SYSTEM TANK_MVCL (* Level Control System Model+View+Control+HMI *)
  (* Standard: 61499-1; Classification: Simulation; ApplicationDomain: Process Control *)
  (* Version 0.4, 2007-08-17, JHC, Holobloc Inc, Added SETUP delays for models & controller, changed AUTO tag to MODE. *)
  (* Version 0.3, 2007-08-15, JHC, Holobloc Inc, Removed space in literal "t#250 ms" *)
  (* Version 0.2, 2007-01-09, JHC, Holobloc Inc, Added tag comments. *)
  (* Version 0.1, 2004-09-13, JHC, Rockwell Automation, Extended from TANK_MVL. *)
  (* Version 0.0, 2004-09-03, JHC, Rockwell Automation, Extended from TANK_MVL. *)
  APPLICATION TANK_CTL (* Tank Control Application *)
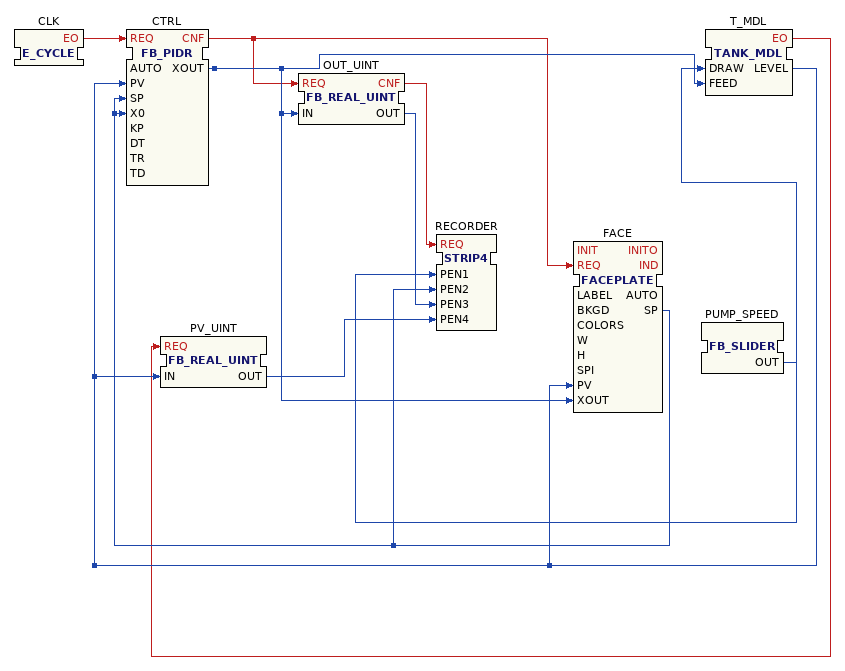
    FBS
      FACE : FACEPLATE;
      CTRL : FB_PIDR;
      RECORDER : STRIP4;
      CLK : E_CYCLE;
      T_MDL : TANK_MDL;
      PUMP_SPEED : FB_SLIDER;
      OUT_UINT : FB_REAL_UINT;
      PV_UINT : FB_REAL_UINT;
    END_FBS
    EVENT_CONNECTIONS
      CLK.EO TO CTRL.REQ;
      CTRL.CNF TO OUT_UINT.REQ;
      T_MDL.EO TO PV_UINT.REQ;
      OUT_UINT.CNF TO RECORDER.REQ;
      CTRL.CNF TO FACE.REQ;
    END_CONNECTIONS
    DATA_CONNECTIONS
      FACE.SP TO CTRL.SP;
      FACE.SP TO CTRL.X0;
      PUMP_SPEED.OUT TO T_MDL.DRAW;
      CTRL.XOUT TO T_MDL.FEED;
      T_MDL.LEVEL TO CTRL.PV;
      T_MDL.LEVEL TO FACE.PV;
      CTRL.XOUT TO FACE.XOUT;
      PUMP_SPEED.OUT TO RECORDER.PEN1;
      FACE.SP TO RECORDER.PEN2;
      CTRL.XOUT TO OUT_UINT.IN;
      OUT_UINT.OUT TO RECORDER.PEN3;
      T_MDL.LEVEL TO PV_UINT.IN;
      PV_UINT.OUT TO RECORDER.PEN4;
    END_CONNECTIONS
  END_APPLICATION
  DEVICE HMI : FRAME_DEVICE(BOUNDS := [240,100,210,270])
    RESOURCE RECORDER : PANEL_RESOURCE
      FBS
        PUMP_SPEED : SUBL_1;
        PV : SUBL_1; (* Measured (Process) Variable *)
        OUT : SUBL_1; (* Manipulated (Output) Variable *)
        RECORDER : STRIP4(COLORS := [red,orange,green,blue], BKGD := COLOR#lightGray, SIZE := [200,150], DX := 1);
        PV_UINT : FB_REAL_UINT;
        OUT_UINT : FB_REAL_UINT;
        SP : SUBL_1; (* Set Point *)
      END_FBS
      EVENT_CONNECTIONS
        PV.IND TO PV_UINT.REQ;
        OUT.IND TO OUT_UINT.REQ;
        START.COLD TO PV.INIT;
        START.WARM TO PV.INIT;
        RECORDER.INITO TO SP.INIT;
        PV.INITO TO PUMP_SPEED.INIT;
        PUMP_SPEED.INITO TO OUT.INIT;
        OUT.INITO TO RECORDER.INIT;
        OUT_UINT.CNF TO RECORDER.REQ;
      END_CONNECTIONS
      DATA_CONNECTIONS
        SP.RD_1 TO RECORDER.PEN2;
        PUMP_SPEED.RD_1 TO RECORDER.PEN1;
        PV.RD_1 TO PV_UINT.IN;
        OUT.RD_1 TO OUT_UINT.IN;
        OUT_UINT.OUT TO RECORDER.PEN3;
        PV_UINT.OUT TO RECORDER.PEN4;
      END_CONNECTIONS
    END_RESOURCE
    RESOURCE PUMP : PANEL_RESOURCE
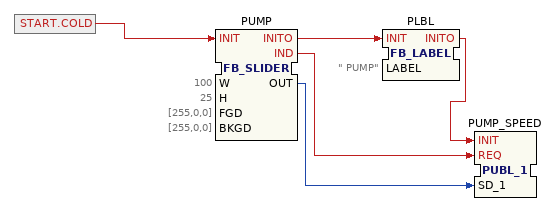
      FBS
        PUMP_SPEED : PUBL_1;
        PUMP : FB_SLIDER(W := 100, H := 25, FGD := [255,0,0], BKGD := [255,0,0]);
        PLBL : FB_LABEL(LABEL := " PUMP");
      END_FBS
      EVENT_CONNECTIONS
        PUMP.INITO TO PLBL.INIT;
        PLBL.INITO TO PUMP_SPEED.INIT;
        START.COLD TO PUMP.INIT;
        PUMP.IND TO PUMP_SPEED.REQ;
      END_CONNECTIONS
      DATA_CONNECTIONS
        PUMP.OUT TO PUMP_SPEED.SD_1;
      END_CONNECTIONS
    END_RESOURCE
  END_DEVICE
  DEVICE CONTROLLER : FRAME_DEVICE(BOUNDS := [100,100,140,270])
    RESOURCE FACE : PANEL_RESOURCE
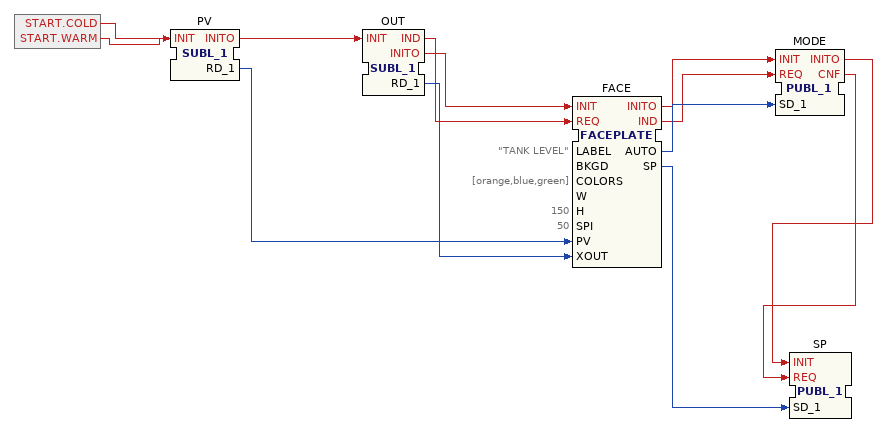
      FBS
        PV : SUBL_1;
        FACE : FACEPLATE(SPI := 50, H := 150, COLORS := [orange,blue,green], LABEL := "TANK LEVEL");
        SP : PUBL_1;
        OUT : SUBL_1;
        MODE : PUBL_1;
      END_FBS
      EVENT_CONNECTIONS
        START.COLD TO PV.INIT;
        START.WARM TO PV.INIT;
        OUT.IND TO FACE.REQ;
        FACE.INITO TO MODE.INIT;
        FACE.IND TO MODE.REQ;
        MODE.INITO TO SP.INIT;
        MODE.CNF TO SP.REQ;
        PV.INITO TO OUT.INIT;
        OUT.INITO TO FACE.INIT;
      END_CONNECTIONS
      DATA_CONNECTIONS
        PV.RD_1 TO FACE.PV;
        FACE.SP TO SP.SD_1;
        OUT.RD_1 TO FACE.XOUT;
        FACE.AUTO TO MODE.SD_1;
      END_CONNECTIONS
    END_RESOURCE
    RESOURCE CTL : EMB_RES
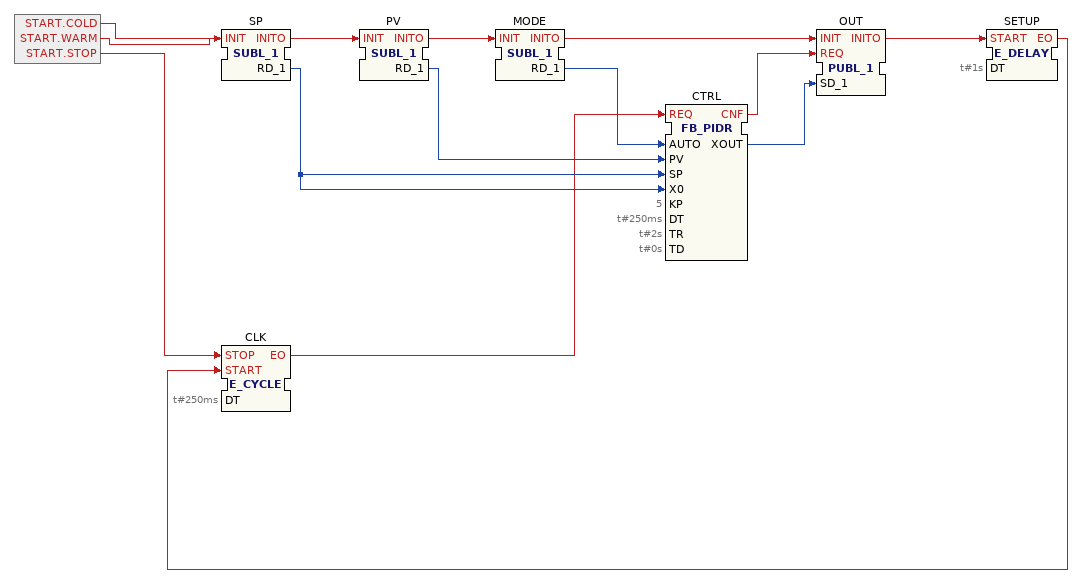
      FBS
        CLK : E_CYCLE(DT := t#250ms);
        PV : SUBL_1;
        SP : SUBL_1;
        CTRL : FB_PIDR(KP := 5, DT := t#250ms, TR := t#2s, TD := t#0s);
        OUT : PUBL_1;
        MODE : SUBL_1; (* 0=Manual, 1=Automatic *)
        SETUP : E_DELAY(DT := t#1s);
      END_FBS
      EVENT_CONNECTIONS
        START.COLD TO SP.INIT;
        START.WARM TO SP.INIT;
        SP.INITO TO PV.INIT;
        PV.INITO TO MODE.INIT;
        MODE.INITO TO OUT.INIT;
        CTRL.CNF TO OUT.REQ;
        CLK.EO TO CTRL.REQ;
        START.STOP TO CLK.STOP;
        OUT.INITO TO SETUP.START;
        SETUP.EO TO CLK.START;
      END_CONNECTIONS
      DATA_CONNECTIONS
        CTRL.XOUT TO OUT.SD_1;
        SP.RD_1 TO CTRL.SP;
        PV.RD_1 TO CTRL.PV;
        MODE.RD_1 TO CTRL.AUTO;
        SP.RD_1 TO CTRL.X0;
      END_CONNECTIONS
    END_RESOURCE
  END_DEVICE
  DEVICE MV : FRAME_DEVICE(BOUNDS := [450,100,175,270]) (* Model+View *)
    RESOURCE TANK_MDL : EMB_RES
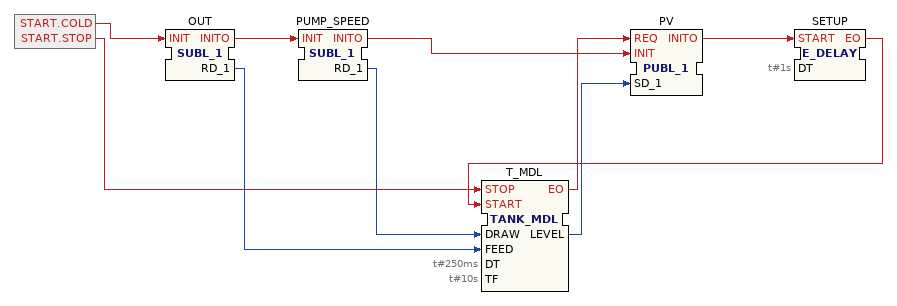
      FBS
        T_MDL : TANK_MDL(DT := t#250ms, TF := t#10s);
        PUMP_SPEED : SUBL_1;
        OUT : SUBL_1;
        PV : PUBL_1;
        SETUP : E_DELAY(DT := t#1s);
      END_FBS
      EVENT_CONNECTIONS
        START.COLD TO OUT.INIT;
        OUT.INITO TO PUMP_SPEED.INIT;
        T_MDL.EO TO PV.REQ;
        START.STOP TO T_MDL.STOP;
        PUMP_SPEED.INITO TO PV.INIT;
        PV.INITO TO SETUP.START;
        SETUP.EO TO T_MDL.START;
      END_CONNECTIONS
      DATA_CONNECTIONS
        PUMP_SPEED.RD_1 TO T_MDL.DRAW;
        OUT.RD_1 TO T_MDL.FEED;
        T_MDL.LEVEL TO PV.SD_1;
      END_CONNECTIONS
    END_RESOURCE
    RESOURCE PUMP_MDL : EMB_RES
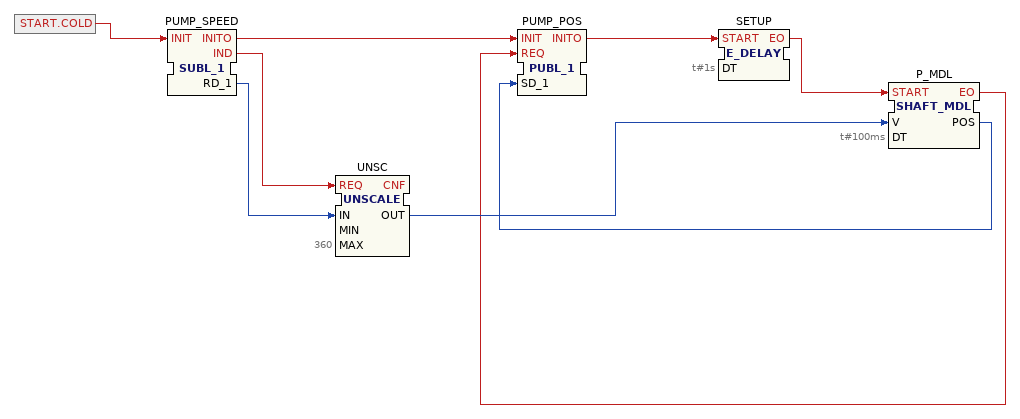
      FBS
        P_MDL : SHAFT_MDL(DT := t#100ms);
        PUMP_POS : PUBL_1;
        PUMP_SPEED : SUBL_1;
        UNSC : UNSCALE(MAX := 360);
        SETUP : E_DELAY(DT := t#1s);
      END_FBS
      EVENT_CONNECTIONS
        START.COLD TO PUMP_SPEED.INIT;
        PUMP_SPEED.INITO TO PUMP_POS.INIT;
        P_MDL.EO TO PUMP_POS.REQ;
        PUMP_SPEED.IND TO UNSC.REQ;
        PUMP_POS.INITO TO SETUP.START;
        SETUP.EO TO P_MDL.START;
      END_CONNECTIONS
      DATA_CONNECTIONS
        P_MDL.POS TO PUMP_POS.SD_1;
        UNSC.OUT TO P_MDL.V;
        PUMP_SPEED.RD_1 TO UNSC.IN;
      END_CONNECTIONS
    END_RESOURCE
    RESOURCE VALVE : VIEW_PANEL(DIA := 50, SIZE := [1,3])
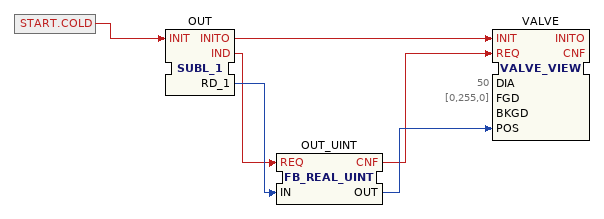
      FBS
        OUT : SUBL_1;
        VALVE : VALVE_VIEW(DIA := 50, FGD := [0,255,0]);
        OUT_UINT : FB_REAL_UINT;
      END_FBS
      EVENT_CONNECTIONS
        START.COLD TO OUT.INIT;
        OUT.INITO TO VALVE.INIT;
        OUT.IND TO OUT_UINT.REQ;
        OUT_UINT.CNF TO VALVE.REQ;
      END_CONNECTIONS
      DATA_CONNECTIONS
        OUT.RD_1 TO OUT_UINT.IN;
        OUT_UINT.OUT TO VALVE.POS;
      END_CONNECTIONS
    END_RESOURCE
    RESOURCE TANK : VIEW_PANEL(SIZE := [1,2], DIA := 75)
      FBS
        TANK : MECH_VIEW(STYLE := VSTYLE#CYLINDER, LEN := 2, DIR := 3, BKGD := [255,255,255], WKPC := [0,0,255]);
        PV : SUBL_1;
        PV_UINT : FB_REAL_UINT;
      END_FBS
      EVENT_CONNECTIONS
        PV.INITO TO TANK.INIT;
        START.COLD TO PV.INIT;
        PV.IND TO PV_UINT.REQ;
        PV_UINT.CNF TO TANK.REQ;
      END_CONNECTIONS
      DATA_CONNECTIONS
        PV.RD_1 TO PV_UINT.IN;
        PV_UINT.OUT TO TANK.POS;
      END_CONNECTIONS
    END_RESOURCE
    RESOURCE PUMP : VIEW_PANEL(DIA := 50, SIZE := [4,1])
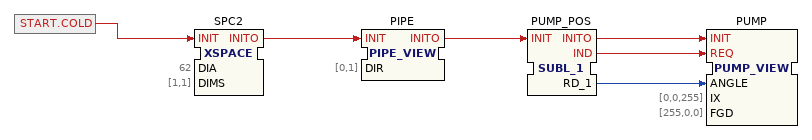
      FBS
        PUMP_POS : SUBL_1;
        SPC2 : XSPACE(DIA := 62, DIMS := [1,1]);
        PIPE : PIPE_VIEW(DIR := [0,1]);
        PUMP : PUMP_VIEW(IX := [0,0,255], FGD := [255,0,0]);
      END_FBS
      EVENT_CONNECTIONS
        SPC2.INITO TO PIPE.INIT;
        START.COLD TO SPC2.INIT;
        PIPE.INITO TO PUMP_POS.INIT;
        PUMP_POS.INITO TO PUMP.INIT;
        PUMP_POS.IND TO PUMP.REQ;
      END_CONNECTIONS
      DATA_CONNECTIONS
        PUMP_POS.RD_1 TO PUMP.ANGLE;
      END_CONNECTIONS
    END_RESOURCE
  END_DEVICE
END_SYSTEM
